{attribute addProperty BoxType "EK1122-0000-0018"}
{attribute addProperty Id "Beckhoff_EPP5xxxsub_EK1100EK1100_179A0949162A_0001_EPP5001_0002_0016EPP5001_99FC62FA13016.25A_0002_EPP5101_0002_0016EPP5101_CA84C7C416220.25A_0003_EPP5101_0002_0017EPP5101_CA84C7C416220.25A_0004_EPP5101_0011_0016EPP5101_19FB32BA16220.25A_0005_EPP5101_0011_0017EPP5101_19FB32BA16220.25A_0006_EPP5101_1002_0016EPP5101_CA84C7C416220.25A_0007_EPP5101_1002_0017EPP5101_CA84C7C416220.25A_0008_EPP5151_0002_0016EPP5151_19FB32BA16220.25A_0009_EPP5151_0002_0017EPP5151_19FB32BA16220.25"}
{attribute addProperty CRC "662546859"}
{attribute addProperty SizeInBites "1442"}
{attribute addProperty SizeInBytes "180.25"}
TYPE Beckhoff_EPP5xxxEK1122_277DA9AB EXTENDS EK1122_179A0949 :
STRUCT
	{attribute addProperty Name "Beckhoff_EPP5xxxsub_EK1100"}
	Beckhoff_EPP5xxxsub_EK1100 : EK1100_179A0949;
	{attribute addProperty Name "A_0001_EPP5001_0002_0016"}
	A_0001_EPP5001_0002_0016 : EPP5001_99FC62FA;
	{attribute addProperty Name "A_0002_EPP5101_0002_0016"}
	A_0002_EPP5101_0002_0016 : EPP5101_CA84C7C4;
	{attribute addProperty Name "A_0003_EPP5101_0002_0017"}
	A_0003_EPP5101_0002_0017 : EPP5101_CA84C7C4;
	{attribute addProperty Name "A_0004_EPP5101_0011_0016"}
	A_0004_EPP5101_0011_0016 : EPP5101_19FB32BA;
	{attribute addProperty Name "A_0005_EPP5101_0011_0017"}
	A_0005_EPP5101_0011_0017 : EPP5101_19FB32BA;
	{attribute addProperty Name "A_0006_EPP5101_1002_0016"}
	A_0006_EPP5101_1002_0016 : EPP5101_CA84C7C4;
	{attribute addProperty Name "A_0007_EPP5101_1002_0017"}
	A_0007_EPP5101_1002_0017 : EPP5101_CA84C7C4;
	{attribute addProperty Name "A_0008_EPP5151_0002_0016"}
	A_0008_EPP5151_0002_0016 : EPP5151_19FB32BA;
	{attribute addProperty Name "A_0009_EPP5151_0002_0017"}
	A_0009_EPP5151_0002_0017 : EPP5151_19FB32BA;
END_STRUCT
END_TYPE

(* stored: Version 1.2.0.0, ProductVersion 3.1.4024.9
   DUT Beckhoff_EPP5xxxEK1122_277DA9AB: Id {f23ed14a-2867-41cc-b9a3-8693fda53701} *)
